(* CODESYS project 42427_Keystone_DeltaICE.project
   Title: 42427_Keystone_DeltaICE
   Description: Delta pick and place with Integrated Case Erector and auto-adjusting cassette. No case sealing, scissor belt exitfeed.
      
      Using PacDrive3 and daisy chained integrated motors, also with one standard drive slice. Festo Ethernet/IP valve banks with input card. Altivar 32 VFDs, 3-Phase is not dropped by safety circuit.
   Version: 0.1.0.0
   Author: Isaac.Brown
   Company: BluePrint Automation

Project tree, tasks and I/O mapping:
  Keystone_DeltaICE : PacDrive LMC 300/400/600C, Schneider Electric, order no. LMCx00C, version 1.51.10.0
    application Application
      task TASK_SR_Main (cyclic, interval t#10ms, priority 31, watchdog t#10ms x 10) calls SR_Main
      program SR_Main [ST]
      SystemSettings/
      Product Codes/
      Collation/
        TYPE/
          data type Collation_typ
        VAR/
          global variables Collation_var
    Message Logger
    EPAS SERCOSIII Device Commissioning
    EPAS Mechatronic
    SERCOSIII : SERCOS III Interface, Schneider Electric, version 1.51.10.0
      PowerSupply : Lexium LXM62 Power Supply, Schneider Electric, order no. LXM62PD84, LXM62PD20, version 1.51.10.0
          settings: ConfiguredApplicationType = 'PSM_Lexium62'
      Ram : Lexium LXM62 Drive, Schneider Electric, order no. LXM62DU60, LXM62DD15, LXM62DD27, LXM62DD45, LXM62DC13, version 1.51.10.0
          settings: ConfiguredApplicationType = 'DRV_Lexium62'
      Delta_A : Lexium ILM62 Drive Module, Schneider Electric, order no. ILM070, ILM100, ILM140, version 1.51.10.0
          settings: ConfiguredApplicationType = 'DRV_ILM62'
      Belt : Lexium LXM62 Drive, Schneider Electric, order no. LXM62DU60, LXM62DD15, LXM62DD27, LXM62DD45, LXM62DC13, version 1.51.10.0
          settings: ConfiguredApplicationType = 'DRV_Lexium62_1'
      Delta_B : Lexium ILM62 Drive Module, Schneider Electric, order no. ILM070, ILM100, ILM140, version 1.51.10.0
          settings: ConfiguredApplicationType = 'DRV_ILM62_1'
      Delta_C : Lexium ILM62 Drive Module, Schneider Electric, order no. ILM070, ILM100, ILM140, version 1.51.10.0
          settings: ConfiguredApplicationType = 'DRV_ILM62_2'
      ICE_A : Lexium ILM62 Drive Module, Schneider Electric, order no. ILM070, ILM100, ILM140, version 1.51.10.0
          settings: ConfiguredApplicationType = 'DRV_ILM62_3'
      ICE_B : Lexium ILM62 Drive Module, Schneider Electric, order no. ILM070, ILM100, ILM140, version 1.51.10.0
          settings: ConfiguredApplicationType = 'DRV_ILM62_4'
      Tipper : Lexium ILM62 Drive Module, Schneider Electric, order no. ILM070, ILM100, ILM140, version 1.51.10.0
          settings: ConfiguredApplicationType = 'DRV_ILM62_5'
      BC_TM5NS31 : TM5NS31, Schneider Electric, order no. TM5NS31, version 1.51.7.0
        TM5SAI4L : TM5SAI4L, Schneider Electric, order no. TM5SAI4L, version 1.51.7.0
            settings: ModuleOk.IDN = 16#040005DF; AnalogInput 0-3.IDN = 16#040005E1; ModuleOk.IDN = 16#040005DF; ModuleOk.Process data out.IDN = 16#00000000; ModuleOk.Process data in.IDN = 16#00000000; ModuleOk.Diag out.IDN = 16#00000000; ModuleOk.Diag in.IDN = 16#041105DF; AnalogInput 0-3.IDN = 16#040005E1; AnalogInput 0-3.Process data out.IDN = 16#00000000; AnalogInput 0-3.Process data in.IDN = 16#040905E1; AnalogInput 0-3.Diag out.IDN = 16#00000000; AnalogInput 0-3.Diag in.IDN = 16#041105E1; PropritaryParameterSet_S-0-1503.0.20.IDN = 16#041405DF
            unmapped channels: ModuleOK, Status Input, AnalogInput 0-3
        TM5SDI2D : TM5SDI2D, Schneider Electric, order no. TM5SDI2D, version 1.35.2.1
            settings: DigitalInput 0-1.IDN = 16#020005DF; DigitalInput 0-1.IDN = 16#020005DF; DigitalInput 0-1.Process data out.IDN = 16#00000000; DigitalInput 0-1.Process data in.IDN = 16#020905DF; DigitalInput 0-1.Diag out.IDN = 16#00000000; DigitalInput 0-1.Diag in.IDN = 16#021105DF; PropritaryParameterSet_S-0-1503.0.20.IDN = 16#021405DF
            unmapped channels: ModuleOK, DigitalInput 0-1
        TM5SPS3 : TM5SPS3, Schneider Electric, order no. TM5SPS3, version 1.50.0.12
            settings: ModuleOk, StatusInput01.IDN = 16#010005DF; SupplyCurrent, SupplyVoltage.IDN = 16#010005E1; ModuleOk, StatusInput01.IDN = 16#010005DF; ModuleOk, StatusInput01.Process data out.IDN = 16#00000000; ModuleOk, StatusInput01.Process data in.IDN = 16#00000000; ModuleOk, StatusInput01.Diag out.IDN = 16#00000000; ModuleOk, StatusInput01.Diag in.IDN = 16#011105DF; SupplyCurrent, SupplyVoltage.IDN = 16#010005E1; SupplyCurrent, SupplyVoltage.Process data out.IDN = 16#00000000; SupplyCurrent, SupplyVoltage.Process data in.IDN = 16#00000000; SupplyCurrent, SupplyVoltage.Diag out.IDN = 16#00000000; SupplyCurrent, SupplyVoltage.Diag in.IDN = 16#011105E1; PropritaryParameterSet_S-0-1503.0.20.IDN = 16#011405DF
            unmapped channels: ModuleOK, DiagIn
        TM5SDI2D_1 : TM5SDI2D, Schneider Electric, order no. TM5SDI2D, version 1.35.2.1
            settings: DigitalInput 0-1.IDN = 16#030005DF; DigitalInput 0-1.IDN = 16#030005DF; DigitalInput 0-1.Process data out.IDN = 16#00000000; DigitalInput 0-1.Process data in.IDN = 16#030905DF; DigitalInput 0-1.Diag out.IDN = 16#00000000; DigitalInput 0-1.Diag in.IDN = 16#031105DF; PropritaryParameterSet_S-0-1503.0.20.IDN = 16#031405DF
            unmapped channels: ModuleOK, DigitalInput 0-1
        TM5SAI4L_1 : TM5SAI4L, Schneider Electric, order no. TM5SAI4L, version 1.51.7.0
            settings: ModuleOk.IDN = 16#050005DF; AnalogInput 0-3.IDN = 16#050005E1; ModuleOk.IDN = 16#050005DF; ModuleOk.Process data out.IDN = 16#00000000; ModuleOk.Process data in.IDN = 16#00000000; ModuleOk.Diag out.IDN = 16#00000000; ModuleOk.Diag in.IDN = 16#051105DF; AnalogInput 0-3.IDN = 16#050005E1; AnalogInput 0-3.Process data out.IDN = 16#00000000; AnalogInput 0-3.Process data in.IDN = 16#050905E1; AnalogInput 0-3.Diag out.IDN = 16#00000000; AnalogInput 0-3.Diag in.IDN = 16#051105E1; PropritaryParameterSet_S-0-1503.0.20.IDN = 16#051405DF
            unmapped channels: ModuleOK, Status Input, AnalogInput 0-3
        TM5SDO12T : TM5SDO12T, Schneider Electric, order no. TM5SDO12T, version 1.35.2.1
            settings: DigitalOutput 1-8, DigitalOutput 9-12.IDN = 16#060005DE; ModuleOk, StatusDigitalOutput 1-8, StatusDigitalOutput 9-12.IDN = 16#060005DF; DigitalOutput 1-8, DigitalOutput 9-12.IDN = 16#060005DE; DigitalOutput 1-8, DigitalOutput 9-12.Process data out.IDN = 16#060505DE; DigitalOutput 1-8, DigitalOutput 9-12.Process data in.IDN = 16#00000000; DigitalOutput 1-8, DigitalOutput 9-12.Diag out.IDN = 16#00000000; DigitalOutput 1-8, DigitalOutput 9-12.Diag in.IDN = 16#00000000; ModuleOk, StatusDigitalOutput 1-8, StatusDigitalOutput 9-12.IDN = 16#060005DF; ModuleOk, StatusDigitalOutput 1-8, StatusDigitalOutput 9-12.Process data out.IDN = 16#00000000; ModuleOk, StatusDigitalOutput 1-8, StatusDigitalOutput 9-12.Process data in.IDN = 16#00000000; ModuleOk, StatusDigitalOutput 1-8, StatusDigitalOutput 9-12.Diag out.IDN = 16#00000000; ModuleOk, StatusDigitalOutput 1-8, StatusDigitalOutput 9-12.Diag in.IDN = 16#061105DF; PropritaryParameterSet_S-0-1503.0.20.IDN = 16#061405DF
            unmapped channels: Outputs, Inputs
        TM5SPS1 : TM5SPS1, Schneider Electric, order no. TM5SPS1, version 1.50.0.12
            settings: ModuleOk, StatusInput01.IDN = 16#070005DF; ModuleOk, StatusInput01.IDN = 16#070005DF; ModuleOk, StatusInput01.Process data out.IDN = 16#00000000; ModuleOk, StatusInput01.Process data in.IDN = 16#00000000; ModuleOk, StatusInput01.Diag out.IDN = 16#00000000; ModuleOk, StatusInput01.Diag in.IDN = 16#071105DF; PropritaryParameterSet_S-0-1503.0.20.IDN = 16#071405DF
            unmapped channels: DiagIn
        TM5SDO12T_1 : TM5SDO12T, Schneider Electric, order no. TM5SDO12T, version 1.35.2.1
            settings: DigitalOutput 1-8, DigitalOutput 9-12.IDN = 16#080005DE; ModuleOk, StatusDigitalOutput 1-8, StatusDigitalOutput 9-12.IDN = 16#080005DF; DigitalOutput 1-8, DigitalOutput 9-12.IDN = 16#080005DE; DigitalOutput 1-8, DigitalOutput 9-12.Process data out.IDN = 16#080505DE; DigitalOutput 1-8, DigitalOutput 9-12.Process data in.IDN = 16#00000000; DigitalOutput 1-8, DigitalOutput 9-12.Diag out.IDN = 16#00000000; DigitalOutput 1-8, DigitalOutput 9-12.Diag in.IDN = 16#00000000; ModuleOk, StatusDigitalOutput 1-8, StatusDigitalOutput 9-12.IDN = 16#080005DF; ModuleOk, StatusDigitalOutput 1-8, StatusDigitalOutput 9-12.Process data out.IDN = 16#00000000; ModuleOk, StatusDigitalOutput 1-8, StatusDigitalOutput 9-12.Process data in.IDN = 16#00000000; ModuleOk, StatusDigitalOutput 1-8, StatusDigitalOutput 9-12.Diag out.IDN = 16#00000000; ModuleOk, StatusDigitalOutput 1-8, StatusDigitalOutput 9-12.Diag in.IDN = 16#081105DF; PropritaryParameterSet_S-0-1503.0.20.IDN = 16#081405DF
            unmapped channels: Outputs, Inputs
    DQG_DigitalOut : Digital Outputs, Schneider Electric, version 1.51.10.0
      DQ_0 : Output, Schneider Electric, version 1.51.10.0
      DQ_1 : Output, Schneider Electric, version 1.51.10.0
      DQ_2 : Output, Schneider Electric, version 1.51.10.0
      DQ_3 : Output, Schneider Electric, version 1.51.10.0
      DQ_4 : Output, Schneider Electric, version 1.51.10.0
      DQ_5 : Output, Schneider Electric, version 1.51.10.0
      DQ_6 : Output, Schneider Electric, version 1.51.10.0
      DQ_7 : Output, Schneider Electric, version 1.51.10.0
      DQ_8 : Output, Schneider Electric, version 1.51.10.0
      DQ_9 : Output, Schneider Electric, version 1.51.10.0
      DQ_10 : Output, Schneider Electric, version 1.51.10.0
      DQ_11 : Output, Schneider Electric, version 1.51.10.0
      DQ_12 : Output, Schneider Electric, version 1.51.10.0
      DQ_13 : Output, Schneider Electric, version 1.51.10.0
      DQ_14 : Output, Schneider Electric, version 1.51.10.0
      DQ_15 : Output, Schneider Electric, version 1.51.10.0
    DIG_DigitalIn : Digital Inputs, Schneider Electric, version 1.51.10.0
      DI_0 : Input, Schneider Electric, version 1.51.10.0
      DI_1 : Input, Schneider Electric, version 1.51.10.0
      DI_2 : Input, Schneider Electric, version 1.51.10.0
      DI_3 : Input, Schneider Electric, version 1.51.10.0
      DI_4 : Input, Schneider Electric, version 1.51.10.0
      DI_5 : Input, Schneider Electric, version 1.51.10.0
      DI_6 : Input, Schneider Electric, version 1.51.10.0
      DI_7 : Input, Schneider Electric, version 1.51.10.0
      DI_8 : Input, Schneider Electric, version 1.51.10.0
      DI_9 : Input, Schneider Electric, version 1.51.10.0
      DI_10 : Input, Schneider Electric, version 1.51.10.0
      DI_11 : Input, Schneider Electric, version 1.51.10.0
      DI_12 : Input, Schneider Electric, version 1.51.10.0
      DI_13 : Input, Schneider Electric, version 1.51.10.0
      DI_14 : Input, Schneider Electric, version 1.51.10.0
      DI_15 : Input, Schneider Electric, version 1.51.10.0
      DI_16 : Input, Schneider Electric, version 1.51.10.0
      DI_17 : Input, Schneider Electric, version 1.51.10.0
      DI_18 : Input, Schneider Electric, version 1.51.10.0
      DI_19 : Input, Schneider Electric, version 1.51.10.0
      FI_0 : Fast Input, Schneider Electric, version 1.51.10.0
      FI_1 : Fast Input, Schneider Electric, version 1.51.10.0
      FI_2 : Fast Input, Schneider Electric, version 1.51.10.0
      FI_3 : Fast Input, Schneider Electric, version 1.51.10.0
    TPG_TPIn : Touch Probe Inputs, Schneider Electric, version 1.51.10.0
      TP_0 : Touch Probe Input, Schneider Electric, version 1.51.10.0
      TP_1 : Touch Probe Input, Schneider Electric, version 1.51.10.0
      TP_2 : Touch Probe Input, Schneider Electric, version 1.51.10.0
      TP_3 : Touch Probe Input, Schneider Electric, version 1.51.10.0
      TP_4 : Touch Probe Input, Schneider Electric, version 1.51.10.0
      TP_5 : Touch Probe Input, Schneider Electric, version 1.51.10.0
      TP_6 : Touch Probe Input, Schneider Electric, version 1.51.10.0
      TP_7 : Touch Probe Input, Schneider Electric, version 1.51.10.0
      TP_8 : Touch Probe Input, Schneider Electric, version 1.51.10.0
      TP_9 : Touch Probe Input, Schneider Electric, version 1.51.10.0
      TP_10 : Touch Probe Input, Schneider Electric, version 1.51.10.0
      TP_11 : Touch Probe Input, Schneider Electric, version 1.51.10.0
      TP_12 : Touch Probe Input, Schneider Electric, version 1.51.10.0
      TP_13 : Touch Probe Input, Schneider Electric, version 1.51.10.0
      TP_14 : Touch Probe Input, Schneider Electric, version 1.51.10.0
      TP_15 : Touch Probe Input, Schneider Electric, version 1.51.10.0
    AI_0 : Analog Input, Schneider Electric, version 1.51.10.0
    AI_1 : Analog Input, Schneider Electric, version 1.51.10.0
    AQ_0 : Analog Output, Schneider Electric, version 1.51.10.0
    AQ_1 : Analog Output, Schneider Electric, version 1.51.10.0
    EIPS_Scanner : EtherNet-IP-Scanner, Schneider Electric, version 1.51.10.0
      Delta_VB : CPX-FB32 Remote IO, Festo AG & Co. KG, order no. CPX-FB32, version Major Revision=16#2, Minor Revision = 16#1
          settings: INITIALIZED = TRUE; IP address of Target = [16#C0,16#A8,16#00,16#02]; Keying.Check Minor Revision = FALSE
      Infeed : ATV32, Schneider Electric, version Major Revision=16#1, Minor Revision = 16#7
          settings: INITIALIZED = TRUE; IP address of Target = [16#C0,16#A8,16#00,16#03]; Keying.Check Minor Revision = FALSE
      CaseFeed : ATV32, Schneider Electric, version Major Revision=16#1, Minor Revision = 16#7
          settings: INITIALIZED = TRUE; IP address of Target = [16#C0,16#A8,16#00,16#04]; Keying.Check Minor Revision = FALSE
      ExitFeed : ATV32, Schneider Electric, version Major Revision=16#1, Minor Revision = 16#7
          settings: INITIALIZED = TRUE; IP address of Target = [16#C0,16#A8,16#00,16#05]; Keying.Check Minor Revision = FALSE
      ICE_VB : CPX-FB32 Remote IO, Festo AG & Co. KG, order no. CPX-FB32, version Major Revision=16#2, Minor Revision = 16#1
          settings: INITIALIZED = TRUE; IP address of Target = [16#C0,16#A8,16#00,16#06]; Keying.Check Minor Revision = FALSE
      Case_VB : CPX-FB32 Remote IO, Festo AG & Co. KG, order no. CPX-FB32, version Major Revision=16#2, Minor Revision = 16#1
          settings: INITIALIZED = TRUE; IP address of Target = [16#C0,16#A8,16#00,16#07]; Keying.Check Minor Revision = FALSE
      AccelBelt : ATV32, Schneider Electric, version Major Revision=16#1, Minor Revision = 16#7
          settings: INITIALIZED = TRUE; IP address of Target = [16#C0,16#A8,16#00,16#08]; Keying.Check Minor Revision = FALSE
  Project Information/
    function GetCompany [ST]
    function GetTitle [ST]
    function GetVersion [ST]
    function GetTextProperty [ST]
    function GetNumberProperty [ST]
    function GetBooleanProperty [ST]
    function GetVersionProperty [ST]
  MainMachine
    PowerSupply
    Ram
      Drive
    Delta_A
      Drive
    Belt
      Drive
    Delta_B
      Drive
    Delta_C
      Drive
    ICE_A
      Drive
    ICE_B
      Drive
    Tipper
      Drive
  MainMachine
    PowerSupply
    Ram
      Drive
    Delta_A
      Drive
    Belt
      Drive
    Delta_B
      Drive
    Delta_C
      Drive
    ICE_A
      Drive
    ICE_B
      Drive
    Tipper
      Drive
*)

// Keystone_DeltaICE/Application/Collation/TYPE/Collation_typ
TYPE 

Collation_typ	:	STRUCT
	TestSTruct	: MyTestStruct_typ;
END_STRUCT

MyTestStruct_typ	:	STRUCT
	SomeBOOL	: BOOL;
END_STRUCT

END_TYPE

// Keystone_DeltaICE/Application/Collation/VAR/Collation_var
VAR_GLOBAL
	
	CollationCon	: Collation_typ;

END_VAR

// Keystone_DeltaICE/Application/SR_Main
PROGRAM SR_Main
VAR
END_VAR

CollationCon.TestSTruct.SomeBOOL:=	1;

END_PROGRAM

// Project Information/GetCompany
// This function has been automatically generated from the project information.
{attribute 'signature_flag' := '1073741824'}
{attribute 'register_in_runtime'}
FUNCTION GetCompany : WSTRING
VAR_INPUT
	
END_VAR

GetCompany := "BluePrint Automation";

END_FUNCTION

// Project Information/GetTitle
// This function has been automatically generated from the project information.
{attribute 'signature_flag' := '1073741824'}
{attribute 'register_in_runtime'}
FUNCTION GetTitle : WSTRING
VAR_INPUT
	
END_VAR

GetTitle := "42427_Keystone_DeltaICE";

END_FUNCTION

// Project Information/GetVersion
// This function has been automatically generated from the project information.
{attribute 'signature_flag' := '1073741824'}
{attribute 'register_in_runtime'}
FUNCTION GetVersion : VERSION
VAR_INPUT
	
END_VAR

GetVersion.uiMajor := 0;
GetVersion.uiMinor := 1;
GetVersion.uiServicePack := 0;
GetVersion.uiPatch := 0;

END_FUNCTION

// Project Information/GetTextProperty
// This function has been automatically generated from the project information.
{attribute 'signature_flag' := '1073741824'}
{attribute 'register_in_runtime'}
FUNCTION GetTextProperty : WSTRING
VAR_INPUT
	stKey: WSTRING;
END_VAR

IF stKey = "Author" THEN
	GetTextProperty := "Isaac.Brown";
ELSIF stKey = "Company" THEN
	GetTextProperty := "BluePrint Automation";
ELSIF stKey = "Description" THEN
	GetTextProperty := "Delta pick and place with Integrated Case Erector and auto-adjusting cassette. No case sealing, scissor belt exitfeed.

Using PacDrive3 and daisy chained integrated motors, also with one standard drive slice. Festo Ethernet/IP valve banks with input card. Altivar 32 VFDs, 3-Phase is not dropped by safety circuit.";
ELSIF stKey = "Project" THEN
	GetTextProperty := "42427_Keystone_DeltaICE";
ELSIF stKey = "Title" THEN
	GetTextProperty := "42427_Keystone_DeltaICE";
ELSE
	GetTextProperty := "";
END_IF

END_FUNCTION

// Project Information/GetNumberProperty
// This function has been automatically generated from the project information.
{attribute 'signature_flag' := '1073741824'}
{attribute 'register_in_runtime'}
FUNCTION GetNumberProperty : DINT
VAR_INPUT
	stKey: WSTRING;
END_VAR

GetNumberProperty := 0;

END_FUNCTION

// Project Information/GetBooleanProperty
// This function has been automatically generated from the project information.
{attribute 'signature_flag' := '1073741824'}
{attribute 'register_in_runtime'}
FUNCTION GetBooleanProperty : BOOL
VAR_INPUT
	stKey: WSTRING;
END_VAR

GetBooleanProperty := FALSE;

END_FUNCTION

// Project Information/GetVersionProperty
// This function has been automatically generated from the project information.
{attribute 'signature_flag' := '1073741824'}
{attribute 'register_in_runtime'}
FUNCTION GetVersionProperty : VERSION
VAR_INPUT
	stKey: WSTRING;
END_VAR

IF stKey = "Version" THEN
	GetVersionProperty.uiMajor := 0;
	GetVersionProperty.uiMinor := 1;
	GetVersionProperty.uiServicePack := 0;
	GetVersionProperty.uiPatch := 0;
ELSE
	GetVersionProperty.uiMajor := 0;
	GetVersionProperty.uiMinor := 0;
	GetVersionProperty.uiServicePack := 0;
	GetVersionProperty.uiPatch := 0;
END_IF

END_FUNCTION
